// TIA Portal V18 export
FUNCTION "AHUTemperatureDemand" : Void   // FC60007, LAD
{ S7_Optimized_Access := 'TRUE' }
VERSION : 0.1
// stored: AutoNumber false, IsIECCheckEnabled false, SetENOAutomatically false, UDAEnableTagReadback false
   VAR_INPUT
      iUnitID : Int;
      cCoolingRegulatorState : Byte;
      cHeatingRegulatorState : Byte;
      rSATActual : Real;
      rSATSP : Real;
      rRATActual : Real;
      rRATSPHeating : Real;
      rRATSPCooling : Real;
   END_VAR
   VAR_OUTPUT
      rHeatingDemand : Real;
      rCoolingDemand : Real;
      rFreshAirTempDemand : Real;
   END_VAR
   VAR_TEMP
      iActualUnitMode_old : Int;
      xResetActualSetpoints : Bool;
   END_VAR
   VAR CONSTANT
      cZero : Byte;
   END_VAR
   VAR_TEMP   // added for the SCL form of the ladder/FBD networks
      _w1 : Bool;
   END_VAR
BEGIN

REGION Network 1: Cooling
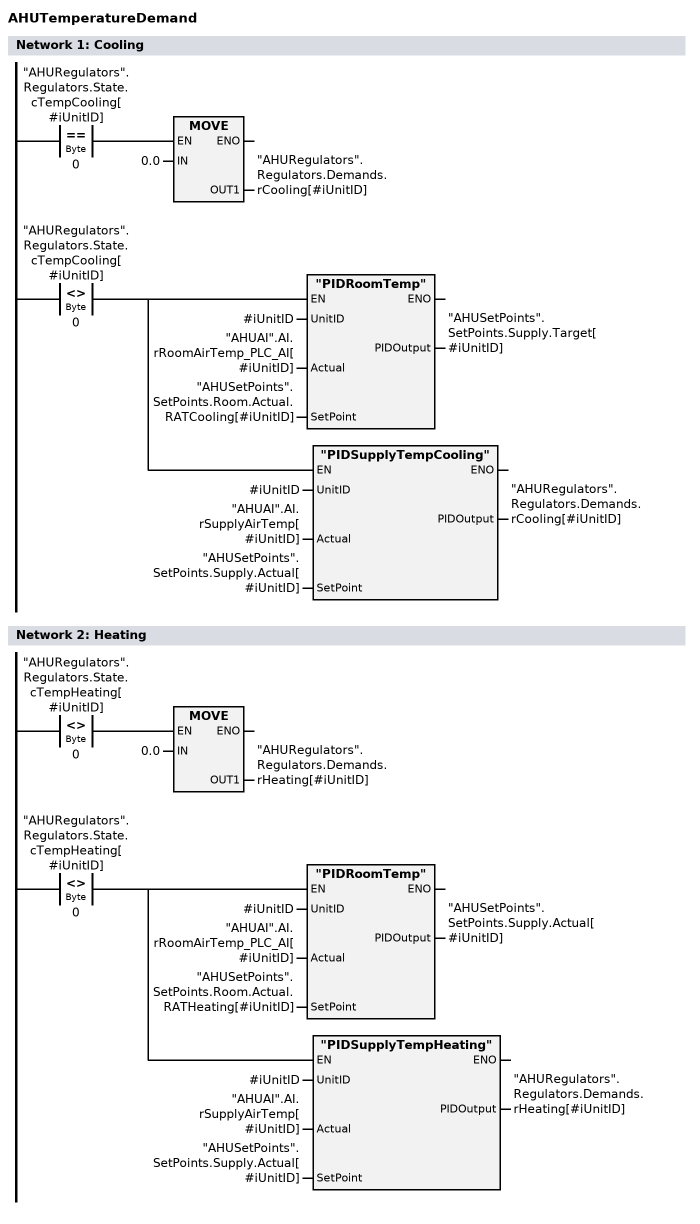
   RUNG wire#powerrail
      { S7_Templates := "SrcType := Byte" } EQ_Contact(in1 := "AHURegulators".Regulators.State.cTempCooling[#iUnitID], in2 := 0)
      Move(in := 0.0, out1 => "AHURegulators".Regulators.Demands.rCooling[#iUnitID])
   END_RUNG
   RUNG wire#powerrail
      { S7_Templates := "SrcType := Byte" } NE_Contact(in1 := "AHURegulators".Regulators.State.cTempCooling[#iUnitID], in2 := 0)
      wire#w1
      "PIDRoomTemp"(UnitID := #iUnitID, Actual := "AHUAI".AI.rRoomAirTemp_PLC_AI[#iUnitID], SetPoint := "AHUSetPoints".SetPoints.Room.Actual.RATCooling[#iUnitID], PIDOutput => "AHUSetPoints".SetPoints.Supply.Target[#iUnitID])
   END_RUNG
   RUNG wire#w1
      "PIDSupplyTempCooling"(UnitID := #iUnitID, Actual := "AHUAI".AI.rSupplyAirTemp[#iUnitID], SetPoint := "AHUSetPoints".SetPoints.Supply.Actual[#iUnitID], PIDOutput => "AHURegulators".Regulators.Demands.rCooling[#iUnitID])
   END_RUNG
   // the same network as SCL:
   IF "AHURegulators".Regulators.State.cTempCooling[#iUnitID] = 0 THEN
       "AHURegulators".Regulators.Demands.rCooling[#iUnitID] := 0.0;
   END_IF;
   #_w1 := "AHURegulators".Regulators.State.cTempCooling[#iUnitID] <> 0;
   IF #_w1 THEN
       "PIDRoomTemp"(UnitID := #iUnitID,
                     Actual := "AHUAI".AI.rRoomAirTemp_PLC_AI[#iUnitID],
                     SetPoint := "AHUSetPoints".SetPoints.Room.Actual.RATCooling[#iUnitID],
                     PIDOutput => "AHUSetPoints".SetPoints.Supply.Target[#iUnitID]);
       "PIDSupplyTempCooling"(UnitID := #iUnitID,
                              Actual := "AHUAI".AI.rSupplyAirTemp[#iUnitID],
                              SetPoint := "AHUSetPoints".SetPoints.Supply.Actual[#iUnitID],
                              PIDOutput => "AHURegulators".Regulators.Demands.rCooling[#iUnitID]);
   END_IF;
END_REGION

REGION Network 2: Heating
   RUNG wire#powerrail
      { S7_Templates := "SrcType := Byte" } NE_Contact(in1 := "AHURegulators".Regulators.State.cTempHeating[#iUnitID], in2 := 0)
      Move(in := 0.0, out1 => "AHURegulators".Regulators.Demands.rHeating[#iUnitID])
   END_RUNG
   RUNG wire#powerrail
      { S7_Templates := "SrcType := Byte" } NE_Contact(in1 := "AHURegulators".Regulators.State.cTempHeating[#iUnitID], in2 := 0)
      wire#w1
      "PIDRoomTemp"(UnitID := #iUnitID, Actual := "AHUAI".AI.rRoomAirTemp_PLC_AI[#iUnitID], SetPoint := "AHUSetPoints".SetPoints.Room.Actual.RATHeating[#iUnitID], PIDOutput => "AHUSetPoints".SetPoints.Supply.Actual[#iUnitID])
   END_RUNG
   RUNG wire#w1
      "PIDSupplyTempHeating"(UnitID := #iUnitID, Actual := "AHUAI".AI.rSupplyAirTemp[#iUnitID], SetPoint := "AHUSetPoints".SetPoints.Supply.Actual[#iUnitID], PIDOutput => "AHURegulators".Regulators.Demands.rHeating[#iUnitID])
   END_RUNG
   // the same network as SCL:
   IF "AHURegulators".Regulators.State.cTempHeating[#iUnitID] <> 0 THEN
       "AHURegulators".Regulators.Demands.rHeating[#iUnitID] := 0.0;
   END_IF;
   #_w1 := "AHURegulators".Regulators.State.cTempHeating[#iUnitID] <> 0;
   IF #_w1 THEN
       "PIDRoomTemp"(UnitID := #iUnitID,
                     Actual := "AHUAI".AI.rRoomAirTemp_PLC_AI[#iUnitID],
                     SetPoint := "AHUSetPoints".SetPoints.Room.Actual.RATHeating[#iUnitID],
                     PIDOutput => "AHUSetPoints".SetPoints.Supply.Actual[#iUnitID]);
       "PIDSupplyTempHeating"(UnitID := #iUnitID,
                              Actual := "AHUAI".AI.rSupplyAirTemp[#iUnitID],
                              SetPoint := "AHUSetPoints".SetPoints.Supply.Actual[#iUnitID],
                              PIDOutput => "AHURegulators".Regulators.Demands.rHeating[#iUnitID]);
   END_IF;
END_REGION
END_FUNCTION
